// TIA Portal project "Level Control" (V14)

(* hardware
DEVICE "S7-1200 station_1"  S7-1200 Station
   slot 0: "Rack_0"  Rack  V1.0
   slot 1: "PLC_1"  CPU 1212C DC/DC/DC  6ES7 212-1AE40-0XB0  V4.2
   slot 2: "AQ 2x14BIT_1"  SM 1232 AQ2  6ES7 232-4HB32-0XB0  V2.0
*)

// ===== PLC "PLC_1"  CPU 1212C DC/DC/DC =====

VAR_GLOBAL   // PLC tag table "Default tag table"
   "Baslat" AT %I0.0 : Bool;
   "baslatma yardimci rolesi" AT %M0.0 : Bool;
   "Analog giris" AT %IW64 : Int;
   "Normalize" AT %MD100 : Real;
   "Analog voltaj" AT %MD200 : DWord;
   "durdurma yardimci rolesi" AT %M0.1 : Bool;
   "Analog cikis" AT %QW96 : Int;
   "Yesil" AT %Q0.1 : Bool;
   "Kirmizi" AT %Q0.2 : Bool;
   "Sari" AT %Q0.0 : Bool;
   "PID2 baslat" AT %I0.1 : Bool;
   "Durdur" AT %I0.2 : Bool;
   "Tag_1" AT %I0.3 : Bool;
   "Manuel_PID yardimci rolesi" AT %M0.2 : Bool;
   "Tag_3" AT %MD2 : DWord;
   "Tag_4" AT %MD3 : DWord;
   "bolunmus voltaj degeri" AT %MD300 : Real;
END_VAR

ORGANIZATION_BLOCK "Sistem"   // OB1, LAD, ProgramCycle
TITLE = "Main Program Sweep (Cycle)"
{ S7_Optimized_Access := 'TRUE' }
VERSION : 0.1
   VAR_INPUT
      Initial_Call : Bool;   // Initial call of this OB
      Remanence : Bool;   // =True, if remanent data are available
   END_VAR
   VAR_TEMP   // added for the SCL form of the ladder/FBD networks
      _w1 : Bool;
   END_VAR
BEGIN

REGION Network 1: PID baslatma durdurma
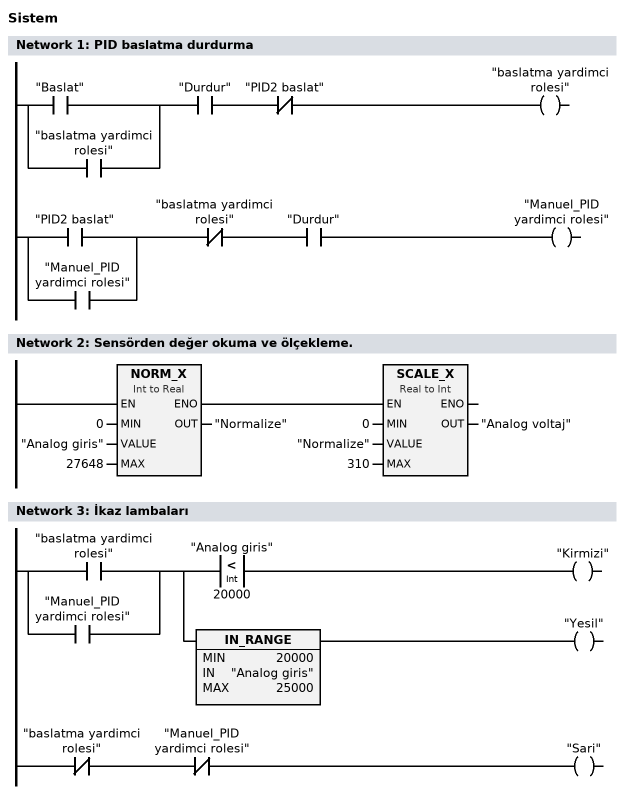
   RUNG wire#powerrail
      Contact( "Baslat" )
      wire#w1
      Contact( "Durdur" )
      I_Contact( "PID2 baslat" )
      Coil( "baslatma yardimci rolesi" )
   END_RUNG
   RUNG wire#powerrail
      Contact( "baslatma yardimci rolesi" )
   END_RUNG wire#w1
   RUNG wire#powerrail
      Contact( "PID2 baslat" )
      wire#w2
      I_Contact( "baslatma yardimci rolesi" )
      Contact( "Durdur" )
      Coil( "Manuel_PID yardimci rolesi" )
   END_RUNG
   RUNG wire#powerrail
      Contact( "Manuel_PID yardimci rolesi" )
   END_RUNG wire#w2
   // the same network as SCL:
   "baslatma yardimci rolesi" := ("Baslat" OR "baslatma yardimci rolesi") AND "Durdur" AND NOT "PID2 baslat";
   "Manuel_PID yardimci rolesi" := ("PID2 baslat" OR "Manuel_PID yardimci rolesi") AND NOT "baslatma yardimci rolesi" AND "Durdur";
END_REGION

REGION Network 2: Sensörden değer okuma ve ölçekleme.
   RUNG wire#powerrail
      { S7_Templates := "[SrcType := Int, DestType := Real]" } Normalize(min := 0, value := "Analog giris", max := 27648, out => "Normalize")
      { S7_Templates := "[SrcType := Real, DestType := Int]" } Scale(min := 0, value := "Normalize", max := 310, out => "Analog voltaj")
   END_RUNG
   // the same network as SCL:
   "Normalize" := NORM_X(MIN := 0, VALUE := "Analog giris", MAX := 27648);
   "Analog voltaj" := SCALE_X(MIN := 0, VALUE := "Normalize", MAX := 310);
END_REGION

REGION Network 3: İkaz lambaları
   RUNG wire#powerrail
      Contact( "baslatma yardimci rolesi" )
      wire#w1
      { S7_Templates := "SrcType := Int" } LT_Contact(in1 := "Analog giris", in2 := 20000)
      Coil( "Kirmizi" )
   END_RUNG
   RUNG wire#powerrail
      Contact( "Manuel_PID yardimci rolesi" )
   END_RUNG wire#w1
   RUNG wire#w1
      { S7_Templates := "SrcType := Int" } InRange(min := 20000, in := "Analog giris", max := 25000)
      Coil( "Yesil" )
   END_RUNG
   RUNG wire#powerrail
      I_Contact( "baslatma yardimci rolesi" )
      I_Contact( "Manuel_PID yardimci rolesi" )
      Coil( "Sari" )
   END_RUNG
   // the same network as SCL:
   #_w1 := "baslatma yardimci rolesi" OR "Manuel_PID yardimci rolesi";
   "Kirmizi" := #_w1 AND ("Analog giris" < 20000);
   "Yesil" := #_w1 AND (20000 <= "Analog giris") AND ("Analog giris" <= 25000);
   "Sari" := NOT "baslatma yardimci rolesi" AND NOT "Manuel_PID yardimci rolesi";
END_REGION
END_ORGANIZATION_BLOCK

ORGANIZATION_BLOCK "PID Kontrol"   // OB30, LAD, CyclicInterrupt
{ S7_Optimized_Access := 'TRUE' }
VERSION : 0.1
   VAR_INPUT
      Initial_Call : Bool;   // Initial call of this OB
      Event_Count : Int;   // Events discarded
   END_VAR
BEGIN

REGION Network 1: PID Blogu
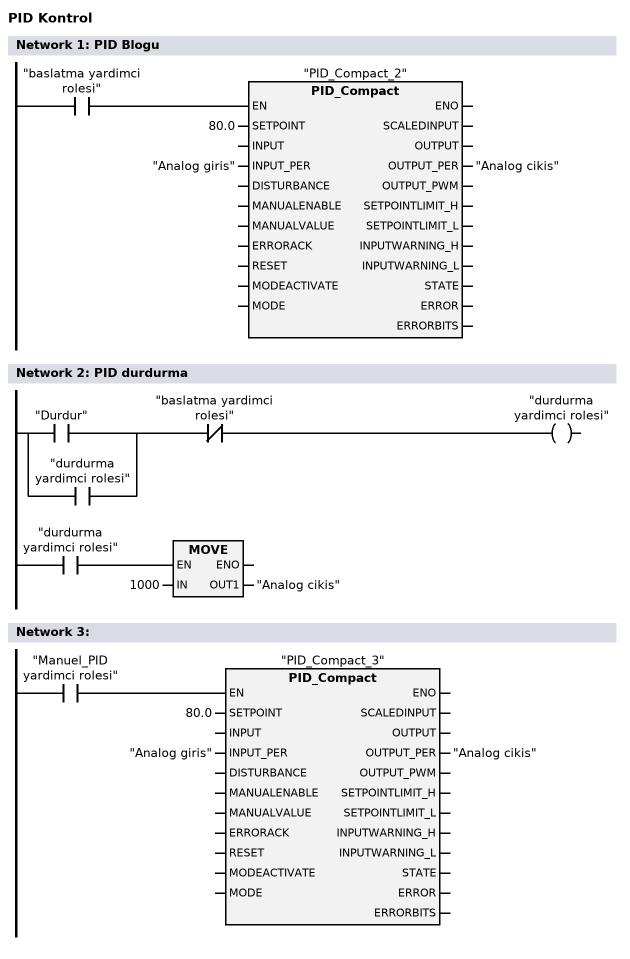
   IF "baslatma yardimci rolesi" THEN
       "PID_Compact_2"(Setpoint := 80.0, Input_PER := "Analog giris", Output_PER => "Analog cikis");   // PID_Compact
   END_IF;
END_REGION

REGION Network 2: PID durdurma
   RUNG wire#powerrail
      Contact( "Durdur" )
      wire#w1
      I_Contact( "baslatma yardimci rolesi" )
      Coil( "durdurma yardimci rolesi" )
   END_RUNG
   RUNG wire#powerrail
      Contact( "durdurma yardimci rolesi" )
   END_RUNG wire#w1
   RUNG wire#powerrail
      Contact( "durdurma yardimci rolesi" )
      Move(in := 1000, out1 => "Analog cikis")
   END_RUNG
   // the same network as SCL:
   "durdurma yardimci rolesi" := ("Durdur" OR "durdurma yardimci rolesi") AND NOT "baslatma yardimci rolesi";
   IF "durdurma yardimci rolesi" THEN "Analog cikis" := 1000; END_IF;
END_REGION

REGION Network 3
   IF "Manuel_PID yardimci rolesi" THEN
       "PID_Compact_3"(Setpoint := 80.0, Input_PER := "Analog giris", Output_PER => "Analog cikis");   // PID_Compact
   END_IF;
END_REGION
END_ORGANIZATION_BLOCK